# EPICS autosave request: RigakuApp/Db/Rigaku_MM003i_settings.req
$(P)$(R)voltage
$(P)$(R)current
